SUBAPPLICATION E_PERMIT_INVERT_3 (* 3-Kanal Invertiertes Event-Freigabe-Gate (F_NOT_BOOL_INIT + E_PERMIT_3) *)
  (* Standard: 61499-2; Description: Copyright (c) 2026 Meisterschulen am Ostbahnhof This program and the accompanying materials are made available under the terms of the Eclipse Public License 2.0 which is available at https://www.eclipse.org/legal/epl-2.0/ SPDX-License-Identifier: EPL-2.0 *)
  (* Version 1.0, 2026-09-10, Franz Höpfinger, Meisterschulen am Ostbahnhof, initial implementation *)
  PACKAGE MyLib::sys;
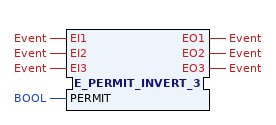
  EVENT_INPUT
    EI1; (* Event input channel 1 *)
    EI2; (* Event input channel 2 *)
    EI3; (* Event input channel 3 *)
  END_EVENT
  EVENT_OUTPUT
    EO1; (* Event output channel 1 *)
    EO2; (* Event output channel 2 *)
    EO3; (* Event output channel 3 *)
  END_EVENT
  VAR_INPUT
    PERMIT : BOOL; (* Invertierte Freigabebedingung *)
  END_VAR
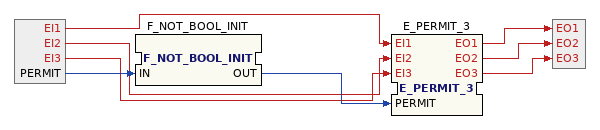
  FBS
    F_NOT_BOOL_INIT : iec61131::booleanOperators::F_NOT_BOOL_INIT;
    E_PERMIT_3 : iec61499::events::E_PERMIT_3;
  END_FBS
  EVENT_CONNECTIONS
    EI1 TO E_PERMIT_3.EI1;
    E_PERMIT_3.EO1 TO EO1;
    EI2 TO E_PERMIT_3.EI2;
    E_PERMIT_3.EO2 TO EO2;
    EI3 TO E_PERMIT_3.EI3;
    E_PERMIT_3.EO3 TO EO3;
  END_CONNECTIONS
  DATA_CONNECTIONS
    PERMIT TO F_NOT_BOOL_INIT.IN;
    F_NOT_BOOL_INIT.OUT TO E_PERMIT_3.PERMIT;
  END_CONNECTIONS
END_SUBAPPLICATION
